// TIA Portal project "Tanque_Acostado" (V15)

(* hardware
DEVICE "S7-1200 station_1"  S7-1200 Station
   slot 0: "Rack_0"  S7-1200 Rack  Rack  V1.0
   slot 1: "PLC_1"  CPU 1214C DC/DC/DC  6ES7 214-1AG40-0XB0  V4.2
*)

// ===== PLC "PLC_1"  CPU 1214C DC/DC/DC =====

VAR_GLOBAL   // PLC tag table "Tabla de variables estándar"
   "Tag_1" AT %IW50 : Int;
   "Altura_H" AT %MD0 : Real;
   "Volumen_tanqueAcostado" AT %MD4 : Real;
END_VAR

ORGANIZATION_BLOCK "Main"   // OB1, LAD, ProgramCycle
TITLE = "Main Program Sweep (Cycle)"
{ S7_Optimized_Access := 'TRUE' }
VERSION : 0.1
   VAR_INPUT
      Initial_Call : Bool;   // Initial call of this OB
      Remanence : Bool;   // =True, if remanent data are available
   END_VAR
   VAR_TEMP
      Convetida1 : Real;
      Diametro : Real;
      Radio : Real;
      Pi : Real;
      Longitud : Real;
      Constante_formula : Real;
   END_VAR
BEGIN

REGION Network 1
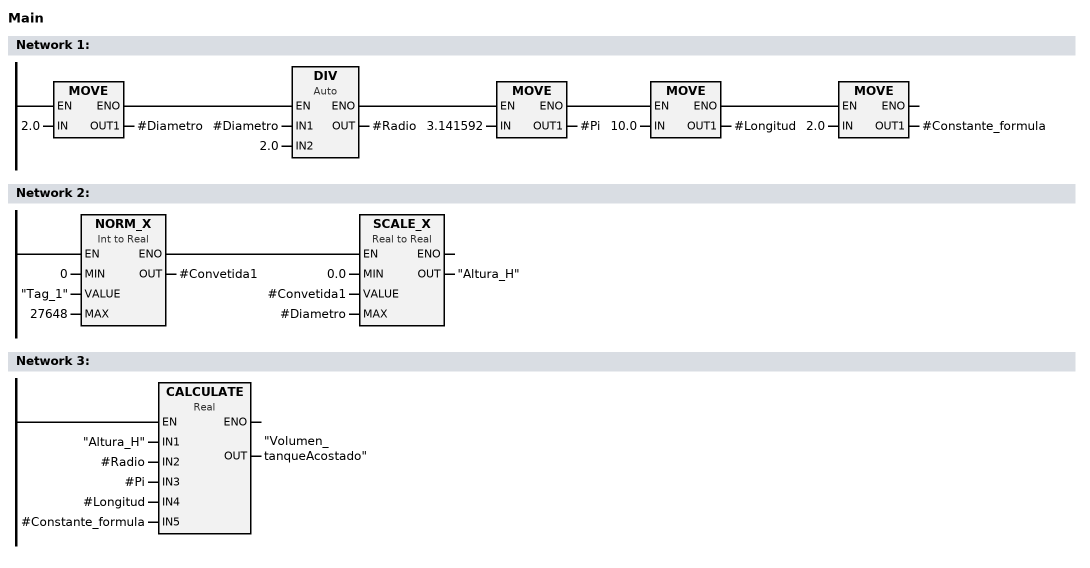
   RUNG wire#powerrail
      Move(in := 2.0, out1 => #Diametro)
      Div(in1 := #Diametro, in2 := 2.0, out => #Radio)
      Move(in := 3.141592, out1 => #Pi)
      Move(in := 10.0, out1 => #Longitud)
      Move(in := 2.0, out1 => #Constante_formula)
   END_RUNG
   // the same network as SCL:
   #Diametro := 2.0;
   #Radio := #Diametro / 2.0;
   #Pi := 3.141592;
   #Longitud := 10.0;
   #Constante_formula := 2.0;
END_REGION

REGION Network 2
   RUNG wire#powerrail
      { S7_Templates := "[SrcType := Int, DestType := Real]" } Normalize(min := 0, value := "Tag_1", max := 27648, out => #Convetida1)
      { S7_Templates := "[SrcType := Real, DestType := Real]" } Scale(min := 0.0, value := #Convetida1, max := #Diametro, out => "Altura_H")
   END_RUNG
   // the same network as SCL:
   #Convetida1 := NORM_X(MIN := 0, VALUE := "Tag_1", MAX := 27648);
   "Altura_H" := SCALE_X(MIN := 0.0, VALUE := #Convetida1, MAX := #Diametro);
END_REGION

REGION Network 3
   RUNG wire#powerrail
      { S7_Templates := "SrcType := Real"; S7_Expression := "IN4 * ((IN3 * SQR(IN2) / IN5) + (IN1 - IN2) * SQRT(IN5 * IN2 * IN1 - SQR(IN1)) + SQR(IN2) * ASIN((-IN2 + IN1) / IN2))" } Calculate(in1 := "Altura_H", in2 := #Radio, in3 := #Pi, in4 := #Longitud, in5 := #Constante_formula, out => "Volumen_tanqueAcostado")
   END_RUNG
   // the same network as SCL:
   "Volumen_tanqueAcostado" := #Longitud * ((#Pi * SQR(#Radio) / #Constante_formula) + ("Altura_H" - #Radio) * SQRT(#Constante_formula * #Radio * "Altura_H" - SQR("Altura_H")) + SQR(#Radio) * ASIN((-#Radio + "Altura_H") / #Radio));
END_REGION
END_ORGANIZATION_BLOCK